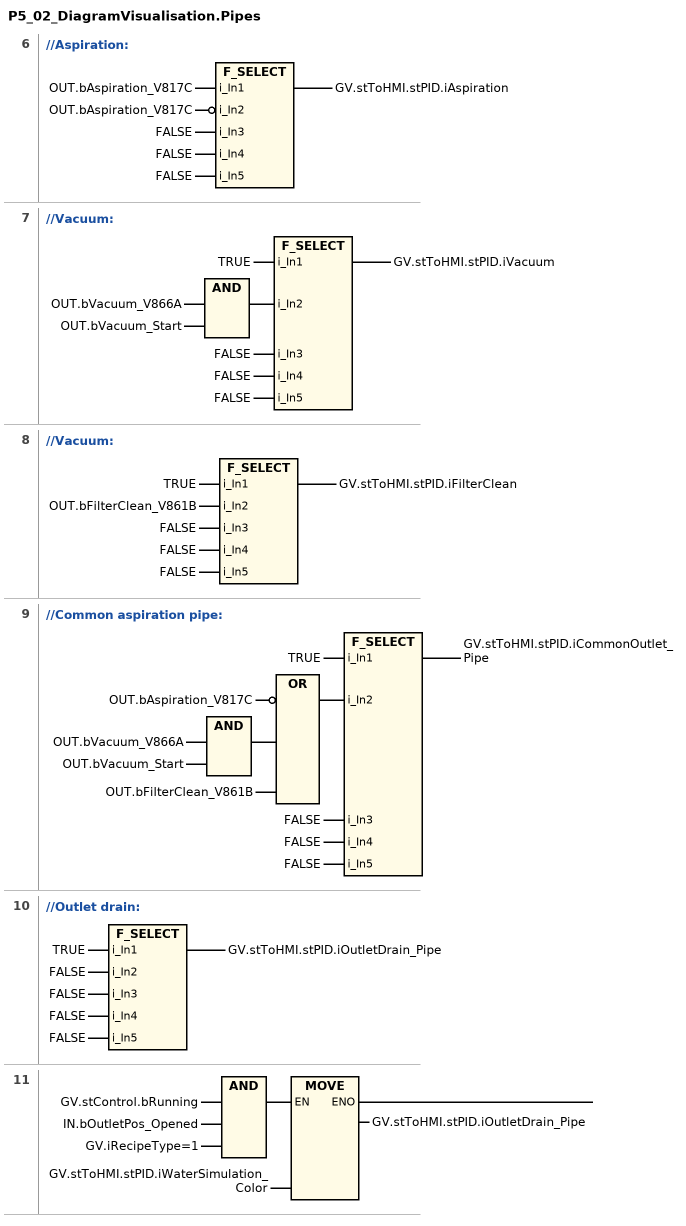
// NETWORK 6
// label: //Aspiration
GV.stToHMI.stPID.iAspiration := F_SELECT(i_In1 := OUT.bAspiration_V817C, i_In2 := NOT OUT.bAspiration_V817C, i_In3 := FALSE, i_In4 := FALSE, i_In5 := FALSE);

// NETWORK 7
// label: //Vacuum
GV.stToHMI.stPID.iVacuum := F_SELECT(i_In1 := TRUE, i_In2 := OUT.bVacuum_V866A AND OUT.bVacuum_Start, i_In3 := FALSE, i_In4 := FALSE, i_In5 := FALSE);

// NETWORK 8
// label: //Vacuum
GV.stToHMI.stPID.iFilterClean := F_SELECT(i_In1 := TRUE, i_In2 := OUT.bFilterClean_V861B, i_In3 := FALSE, i_In4 := FALSE, i_In5 := FALSE);

// NETWORK 9
// label: //Common aspiration pipe
GV.stToHMI.stPID.iCommonOutlet_Pipe := F_SELECT(i_In1 := TRUE, i_In2 := NOT OUT.bAspiration_V817C OR OUT.bVacuum_V866A AND OUT.bVacuum_Start OR OUT.bFilterClean_V861B, i_In3 := FALSE, i_In4 := FALSE, i_In5 := FALSE);

// NETWORK 10
// label: //Outlet drain
GV.stToHMI.stPID.iOutletDrain_Pipe := F_SELECT(i_In1 := TRUE, i_In2 := FALSE, i_In3 := FALSE, i_In4 := FALSE, i_In5 := FALSE);

// NETWORK 11
IF GV.stControl.bRunning AND IN.bOutletPos_Opened AND (GV.iRecipeType=1) THEN
    GV.stToHMI.stPID.iOutletDrain_Pipe := GV.stToHMI.stPID.iWaterSimulation_Color;
END_IF

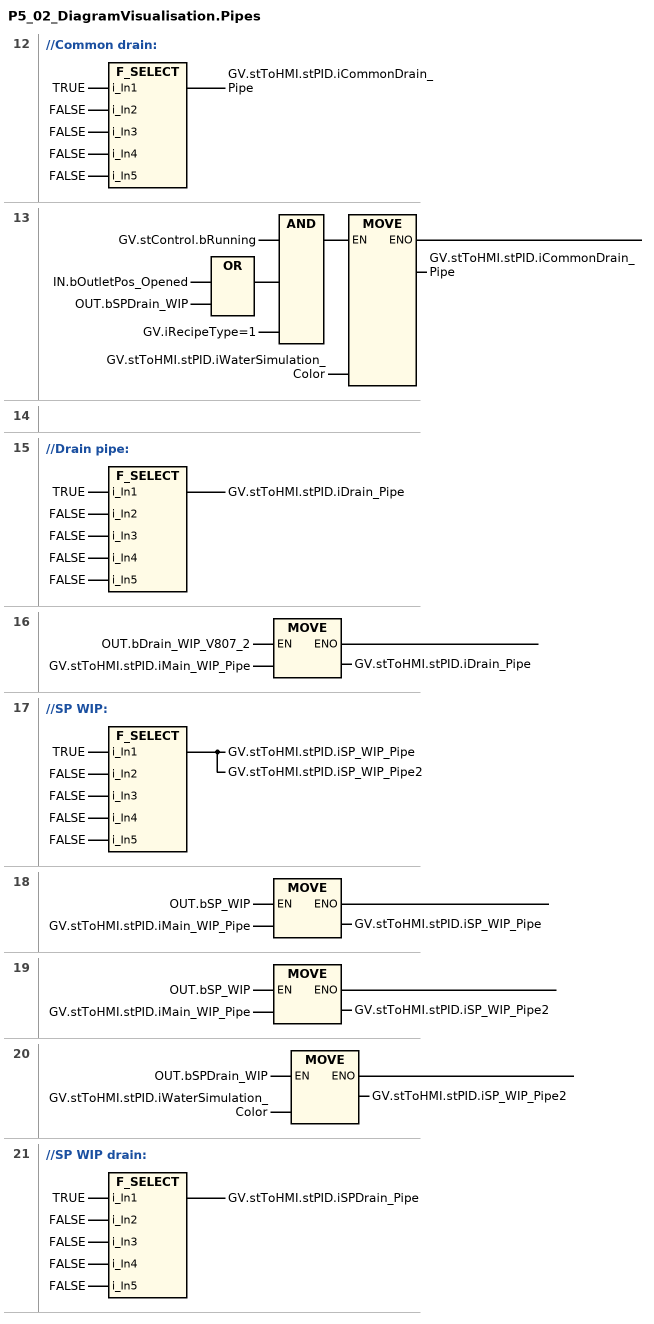
// NETWORK 12
// label: //Common drain
GV.stToHMI.stPID.iCommonDrain_Pipe := F_SELECT(i_In1 := TRUE, i_In2 := FALSE, i_In3 := FALSE, i_In4 := FALSE, i_In5 := FALSE);

// NETWORK 13
IF GV.stControl.bRunning AND (IN.bOutletPos_Opened OR OUT.bSPDrain_WIP) AND (GV.iRecipeType=1) THEN
    GV.stToHMI.stPID.iCommonDrain_Pipe := GV.stToHMI.stPID.iWaterSimulation_Color;
END_IF

// NETWORK 14

// NETWORK 15
// label: //Drain pipe
GV.stToHMI.stPID.iDrain_Pipe := F_SELECT(i_In1 := TRUE, i_In2 := FALSE, i_In3 := FALSE, i_In4 := FALSE, i_In5 := FALSE);

// NETWORK 16
IF OUT.bDrain_WIP_V807_2 THEN GV.stToHMI.stPID.iDrain_Pipe := GV.stToHMI.stPID.iMain_WIP_Pipe; END_IF

// NETWORK 17
// label: //SP WIP
_w4 := F_SELECT(i_In1 := TRUE, i_In2 := FALSE, i_In3 := FALSE, i_In4 := FALSE, i_In5 := FALSE);
GV.stToHMI.stPID.iSP_WIP_Pipe := _w4;
GV.stToHMI.stPID.iSP_WIP_Pipe2 := _w4;

// NETWORK 18
IF OUT.bSP_WIP THEN GV.stToHMI.stPID.iSP_WIP_Pipe := GV.stToHMI.stPID.iMain_WIP_Pipe; END_IF

// NETWORK 19
IF OUT.bSP_WIP THEN GV.stToHMI.stPID.iSP_WIP_Pipe2 := GV.stToHMI.stPID.iMain_WIP_Pipe; END_IF

// NETWORK 20
IF OUT.bSPDrain_WIP THEN GV.stToHMI.stPID.iSP_WIP_Pipe2 := GV.stToHMI.stPID.iWaterSimulation_Color; END_IF

// NETWORK 21
// label: //SP WIP drain
GV.stToHMI.stPID.iSPDrain_Pipe := F_SELECT(i_In1 := TRUE, i_In2 := FALSE, i_In3 := FALSE, i_In4 := FALSE, i_In5 := FALSE);

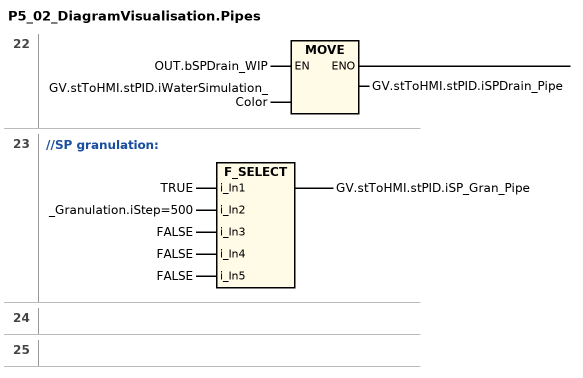
// NETWORK 22
IF OUT.bSPDrain_WIP THEN GV.stToHMI.stPID.iSPDrain_Pipe := GV.stToHMI.stPID.iWaterSimulation_Color; END_IF

// NETWORK 23
// label: //SP granulation
GV.stToHMI.stPID.iSP_Gran_Pipe := F_SELECT(i_In1 := TRUE, i_In2 := _Granulation.iStep=500, i_In3 := FALSE, i_In4 := FALSE, i_In5 := FALSE);

// NETWORK 24

// NETWORK 25
END_ACTION

ACTION Sensors:
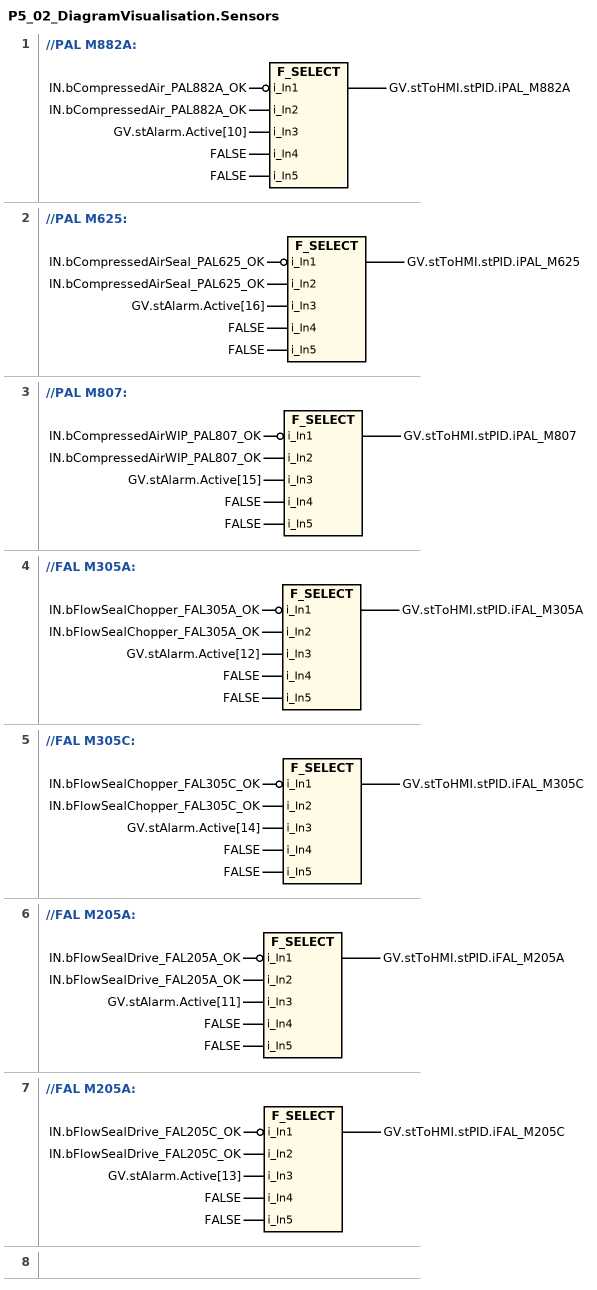
// NETWORK 1
// label: //PAL M882A
GV.stToHMI.stPID.iPAL_M882A := F_SELECT(i_In1 := NOT IN.bCompressedAir_PAL882A_OK, i_In2 := IN.bCompressedAir_PAL882A_OK, i_In3 := GV.stAlarm.Active[10], i_In4 := FALSE, i_In5 := FALSE);

// NETWORK 2
// label: //PAL M625
GV.stToHMI.stPID.iPAL_M625 := F_SELECT(i_In1 := NOT IN.bCompressedAirSeal_PAL625_OK, i_In2 := IN.bCompressedAirSeal_PAL625_OK, i_In3 := GV.stAlarm.Active[16], i_In4 := FALSE, i_In5 := FALSE);

// NETWORK 3
// label: //PAL M807
GV.stToHMI.stPID.iPAL_M807 := F_SELECT(i_In1 := NOT IN.bCompressedAirWIP_PAL807_OK, i_In2 := IN.bCompressedAirWIP_PAL807_OK, i_In3 := GV.stAlarm.Active[15], i_In4 := FALSE, i_In5 := FALSE);

// NETWORK 4
// label: //FAL M305A
GV.stToHMI.stPID.iFAL_M305A := F_SELECT(i_In1 := NOT IN.bFlowSealChopper_FAL305A_OK, i_In2 := IN.bFlowSealChopper_FAL305A_OK, i_In3 := GV.stAlarm.Active[12], i_In4 := FALSE, i_In5 := FALSE);

// NETWORK 5
// label: //FAL M305C
GV.stToHMI.stPID.iFAL_M305C := F_SELECT(i_In1 := NOT IN.bFlowSealChopper_FAL305C_OK, i_In2 := IN.bFlowSealChopper_FAL305C_OK, i_In3 := GV.stAlarm.Active[14], i_In4 := FALSE, i_In5 := FALSE);

// NETWORK 6
// label: //FAL M205A
GV.stToHMI.stPID.iFAL_M205A := F_SELECT(i_In1 := NOT IN.bFlowSealDrive_FAL205A_OK, i_In2 := IN.bFlowSealDrive_FAL205A_OK, i_In3 := GV.stAlarm.Active[11], i_In4 := FALSE, i_In5 := FALSE);

// NETWORK 7
// label: //FAL M205A
GV.stToHMI.stPID.iFAL_M205C := F_SELECT(i_In1 := NOT IN.bFlowSealDrive_FAL205C_OK, i_In2 := IN.bFlowSealDrive_FAL205C_OK, i_In3 := GV.stAlarm.Active[13], i_In4 := FALSE, i_In5 := FALSE);

// NETWORK 8
END_ACTION

ACTION Units:
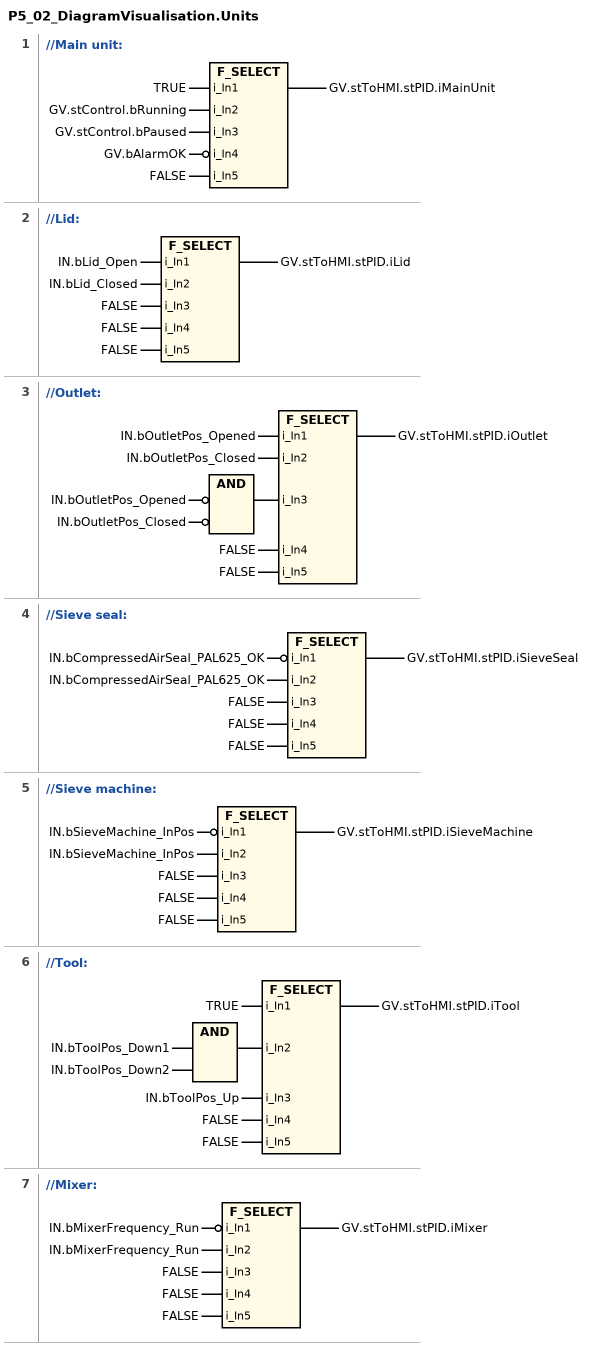
// NETWORK 1
// label: //Main unit
GV.stToHMI.stPID.iMainUnit := F_SELECT(i_In1 := TRUE, i_In2 := GV.stControl.bRunning, i_In3 := GV.stControl.bPaused, i_In4 := NOT GV.bAlarmOK, i_In5 := FALSE);

// NETWORK 2
// label: //Lid
GV.stToHMI.stPID.iLid := F_SELECT(i_In1 := IN.bLid_Open, i_In2 := IN.bLid_Closed, i_In3 := FALSE, i_In4 := FALSE, i_In5 := FALSE);

// NETWORK 3
// label: //Outlet
GV.stToHMI.stPID.iOutlet := F_SELECT(i_In1 := IN.bOutletPos_Opened, i_In2 := IN.bOutletPos_Closed, i_In3 := NOT IN.bOutletPos_Opened AND NOT IN.bOutletPos_Closed, i_In4 := FALSE, i_In5 := FALSE);

// NETWORK 4
// label: //Sieve seal
GV.stToHMI.stPID.iSieveSeal := F_SELECT(i_In1 := NOT IN.bCompressedAirSeal_PAL625_OK, i_In2 := IN.bCompressedAirSeal_PAL625_OK, i_In3 := FALSE, i_In4 := FALSE, i_In5 := FALSE);

// NETWORK 5
// label: //Sieve machine
GV.stToHMI.stPID.iSieveMachine := F_SELECT(i_In1 := NOT IN.bSieveMachine_InPos, i_In2 := IN.bSieveMachine_InPos, i_In3 := FALSE, i_In4 := FALSE, i_In5 := FALSE);

// NETWORK 6
// label: //Tool
GV.stToHMI.stPID.iTool := F_SELECT(i_In1 := TRUE, i_In2 := IN.bToolPos_Down1 AND IN.bToolPos_Down2, i_In3 := IN.bToolPos_Up, i_In4 := FALSE, i_In5 := FALSE);

// NETWORK 7
// label: //Mixer
GV.stToHMI.stPID.iMixer := F_SELECT(i_In1 := NOT IN.bMixerFrequency_Run, i_In2 := IN.bMixerFrequency_Run, i_In3 := FALSE, i_In4 := FALSE, i_In5 := FALSE);

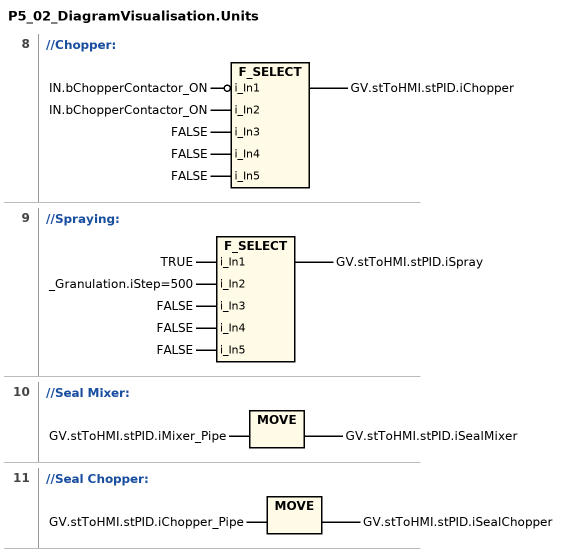
// NETWORK 8
// label: //Chopper
GV.stToHMI.stPID.iChopper := F_SELECT(i_In1 := NOT IN.bChopperContactor_ON, i_In2 := IN.bChopperContactor_ON, i_In3 := FALSE, i_In4 := FALSE, i_In5 := FALSE);

// NETWORK 9
// label: //Spraying
GV.stToHMI.stPID.iSpray := F_SELECT(i_In1 := TRUE, i_In2 := _Granulation.iStep=500, i_In3 := FALSE, i_In4 := FALSE, i_In5 := FALSE);

// NETWORK 10
// label: //Seal Mixer
GV.stToHMI.stPID.iSealMixer := GV.stToHMI.stPID.iMixer_Pipe;

// NETWORK 11
// label: //Seal Chopper
GV.stToHMI.stPID.iSealChopper := GV.stToHMI.stPID.iChopper_Pipe;
END_ACTION

END_PROGRAM

// ---- Functions/F_Select.TcPOU
FUNCTION F_Select : INT
VAR_INPUT
	i_In1			:BOOL;
	i_In2			:BOOL;
	i_In3			:BOOL;
	i_In4			:BOOL;
	i_In5			:BOOL;
END_VAR
VAR
END_VAR

IF i_In1 THEN
	F_Select:=0;
END_IF
IF i_In2 THEN
	F_Select:=1;
END_IF
IF i_In3 THEN
	F_Select:=2;
END_IF
IF i_In4 THEN
	F_Select:=3;
END_IF
IF i_In5 THEN
	F_Select:=4;
END_IF

END_FUNCTION

// ---- POUs/5. HMI/P5_03_OtherControl.TcPOU
PROGRAM P5_03_OtherControl
VAR
	iSeqControl				:INT;
	tSubStepET				:TIME;
	tSubStepPT				:TIME;
	iSubStepMC				:INT;
	iSubStepPC				:INT;
END_VAR
VAR // added by the converter: edge detectors and wires of the graphical bodies
    _w1, _w2 : TIME;
    _w3, _w4 : BOOL;
END_VAR

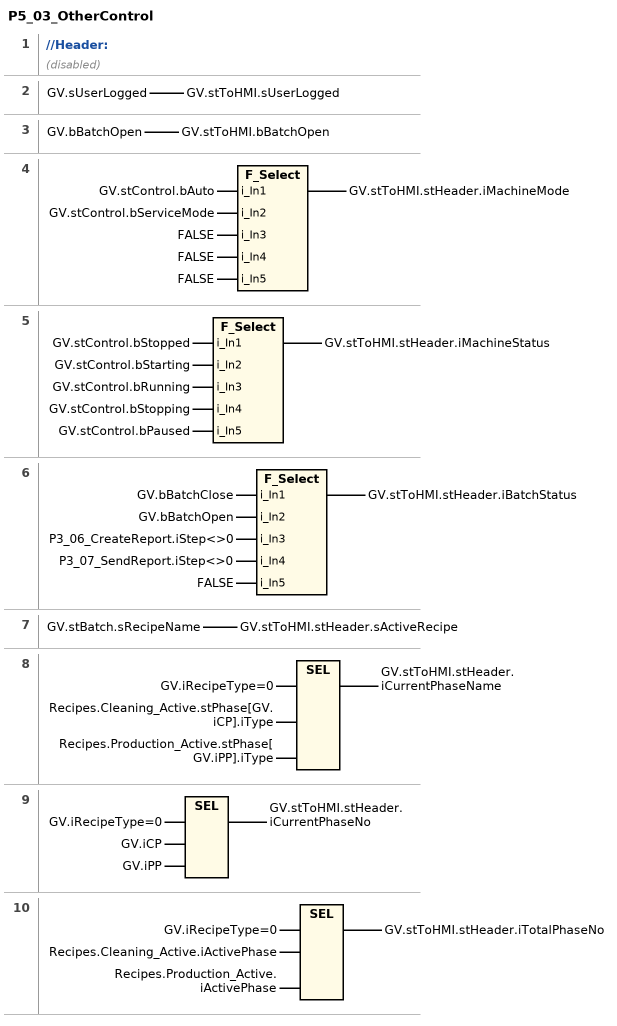
// NETWORK 1 (disabled)
// label: //Header

// NETWORK 2
GV.stToHMI.sUserLogged := GV.sUserLogged;

// NETWORK 3
GV.stToHMI.bBatchOpen := GV.bBatchOpen;

// NETWORK 4
GV.stToHMI.stHeader.iMachineMode := F_Select(i_In1 := GV.stControl.bAuto, i_In2 := GV.stControl.bServiceMode, i_In3 := FALSE, i_In4 := FALSE, i_In5 := FALSE);

// NETWORK 5
GV.stToHMI.stHeader.iMachineStatus := F_Select(i_In1 := GV.stControl.bStopped, i_In2 := GV.stControl.bStarting, i_In3 := GV.stControl.bRunning, i_In4 := GV.stControl.bStopping, i_In5 := GV.stControl.bPaused);

// NETWORK 6
GV.stToHMI.stHeader.iBatchStatus := F_Select(i_In1 := GV.bBatchClose, i_In2 := GV.bBatchOpen, i_In3 := P3_06_CreateReport.iStep<>0, i_In4 := P3_07_SendReport.iStep<>0, i_In5 := FALSE);

// NETWORK 7
GV.stToHMI.stHeader.sActiveRecipe := GV.stBatch.sRecipeName;

// NETWORK 8
GV.stToHMI.stHeader.iCurrentPhaseName := SEL(GV.iRecipeType=0, Recipes.Cleaning_Active.stPhase[GV.iCP].iType, Recipes.Production_Active.stPhase[GV.iPP].iType);

// NETWORK 9
GV.stToHMI.stHeader.iCurrentPhaseNo := SEL(GV.iRecipeType=0, GV.iCP, GV.iPP);

// NETWORK 10
GV.stToHMI.stHeader.iTotalPhaseNo := SEL(GV.iRecipeType=0, Recipes.Cleaning_Active.iActivePhase, Recipes.Production_Active.iActivePhase);

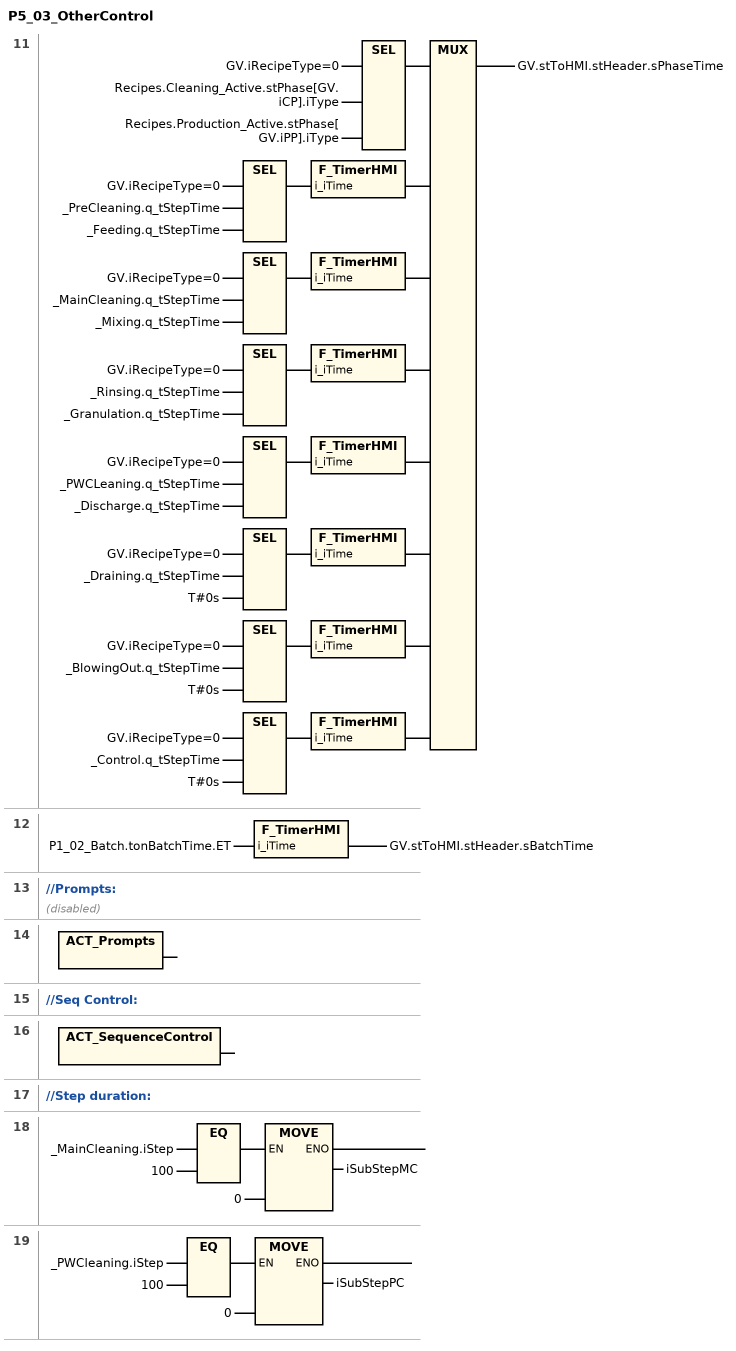
// NETWORK 11
GV.stToHMI.stHeader.sPhaseTime := MUX(SEL(GV.iRecipeType=0, Recipes.Cleaning_Active.stPhase[GV.iCP].iType, Recipes.Production_Active.stPhase[GV.iPP].iType), F_TimerHMI(i_iTime := SEL(GV.iRecipeType=0, _PreCleaning.q_tStepTime, _Feeding.q_tStepTime)), F_TimerHMI(i_iTime := SEL(GV.iRecipeType=0, _MainCleaning.q_tStepTime, _Mixing.q_tStepTime)), F_TimerHMI(i_iTime := SEL(GV.iRecipeType=0, _Rinsing.q_tStepTime, _Granulation.q_tStepTime)), F_TimerHMI(i_iTime := SEL(GV.iRecipeType=0, _PWCLeaning.q_tStepTime, _Discharge.q_tStepTime)), F_TimerHMI(i_iTime := SEL(GV.iRecipeType=0, _Draining.q_tStepTime, T#0s)), F_TimerHMI(i_iTime := SEL(GV.iRecipeType=0, _BlowingOut.q_tStepTime, T#0s)), F_TimerHMI(i_iTime := SEL(GV.iRecipeType=0, _Control.q_tStepTime, T#0s)));

// NETWORK 12
GV.stToHMI.stHeader.sBatchTime := F_TimerHMI(i_iTime := P1_02_Batch.tonBatchTime.ET);

// NETWORK 13 (disabled)
// label: //Prompts

// NETWORK 14
ACT_Prompts();

// NETWORK 15
// label: //Seq Control

// NETWORK 16
ACT_SequenceControl();

// NETWORK 17
// label: //Step duration

// NETWORK 18
IF _MainCleaning.iStep = 100 THEN iSubStepMC := 0; END_IF

// NETWORK 19
IF _PWCleaning.iStep = 100 THEN iSubStepPC := 0; END_IF

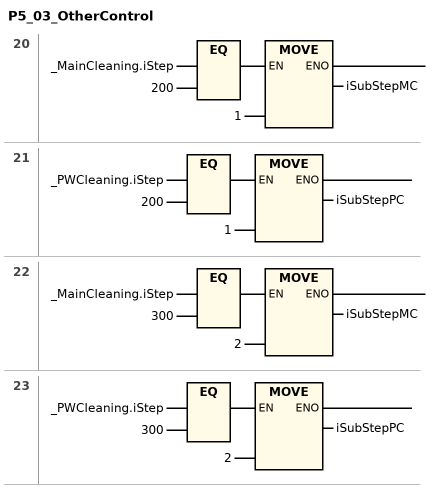
// NETWORK 20
IF _MainCleaning.iStep = 200 THEN iSubStepMC := 1; END_IF

// NETWORK 21
IF _PWCleaning.iStep = 200 THEN iSubStepPC := 1; END_IF

// NETWORK 22
IF _MainCleaning.iStep = 300 THEN iSubStepMC := 2; END_IF

// NETWORK 23
IF _PWCleaning.iStep = 300 THEN iSubStepPC := 2; END_IF

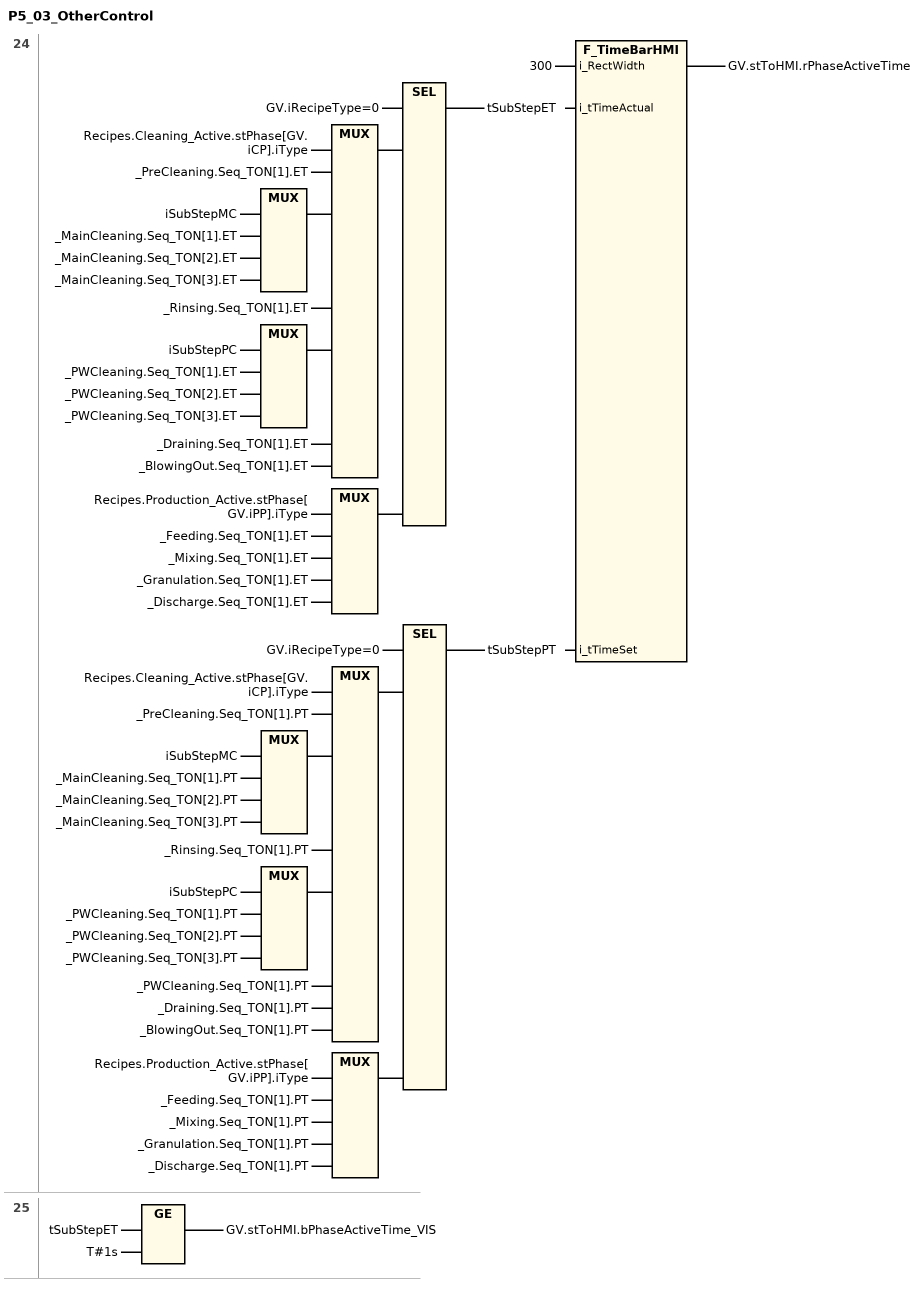
// NETWORK 24
_w1 := SEL(GV.iRecipeType=0, MUX(Recipes.Cleaning_Active.stPhase[GV.iCP].iType, _PreCleaning.Seq_TON[1].ET, MUX(iSubStepMC, _MainCleaning.Seq_TON[1].ET, _MainCleaning.Seq_TON[2].ET, _MainCleaning.Seq_TON[3].ET), _Rinsing.Seq_TON[1].ET, MUX(iSubStepPC, _PWCleaning.Seq_TON[1].ET, _PWCleaning.Seq_TON[2].ET, _PWCleaning.Seq_TON[3].ET), _Draining.Seq_TON[1].ET, _BlowingOut.Seq_TON[1].ET), MUX(Recipes.Production_Active.stPhase[GV.iPP].iType, _Feeding.Seq_TON[1].ET, _Mixing.Seq_TON[1].ET, _Granulation.Seq_TON[1].ET, _Discharge.Seq_TON[1].ET));
tSubStepET := _w1;
_w2 := SEL(GV.iRecipeType=0, MUX(Recipes.Cleaning_Active.stPhase[GV.iCP].iType, _PreCleaning.Seq_TON[1].PT, MUX(iSubStepMC, _MainCleaning.Seq_TON[1].PT, _MainCleaning.Seq_TON[2].PT, _MainCleaning.Seq_TON[3].PT), _Rinsing.Seq_TON[1].PT, MUX(iSubStepPC, _PWCleaning.Seq_TON[1].PT, _PWCleaning.Seq_TON[2].PT, _PWCleaning.Seq_TON[3].PT), _PWCleaning.Seq_TON[1].PT, _Draining.Seq_TON[1].PT, _BlowingOut.Seq_TON[1].PT), MUX(Recipes.Production_Active.stPhase[GV.iPP].iType, _Feeding.Seq_TON[1].PT, _Mixing.Seq_TON[1].PT, _Granulation.Seq_TON[1].PT, _Discharge.Seq_TON[1].PT));
tSubStepPT := _w2;
GV.stToHMI.rPhaseActiveTime := F_TimeBarHMI(i_RectWidth := 300, i_tTimeActual := _w1, i_tTimeSet := _w2);

// NETWORK 25
GV.stToHMI.bPhaseActiveTime_VIS := tSubStepET >= T#1s;

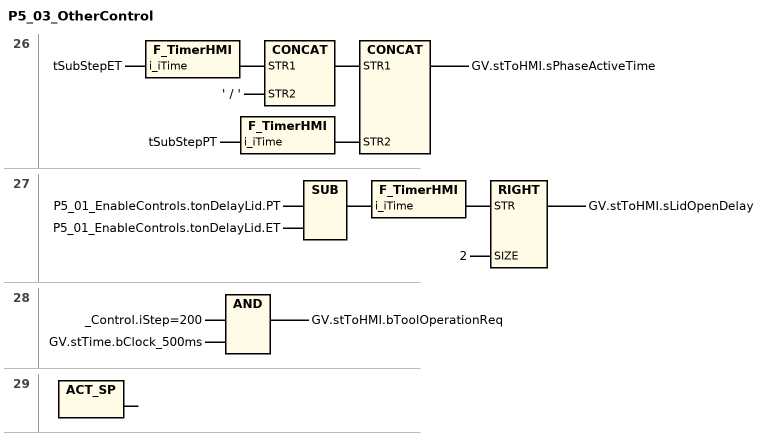
// NETWORK 26
GV.stToHMI.sPhaseActiveTime := CONCAT(STR1 := CONCAT(STR1 := F_TimerHMI(i_iTime := tSubStepET), STR2 := ' / '), STR2 := F_TimerHMI(i_iTime := tSubStepPT));

// NETWORK 27
GV.stToHMI.sLidOpenDelay := RIGHT(STR := F_TimerHMI(i_iTime := P5_01_EnableControls.tonDelayLid.PT - P5_01_EnableControls.tonDelayLid.ET), SIZE := 2);

// NETWORK 28
GV.stToHMI.bToolOperationReq := (_Control.iStep=200) AND GV.stTime.bClock_500ms;

// NETWORK 29
ACT_SP();

ACTION ACT_Prompts:
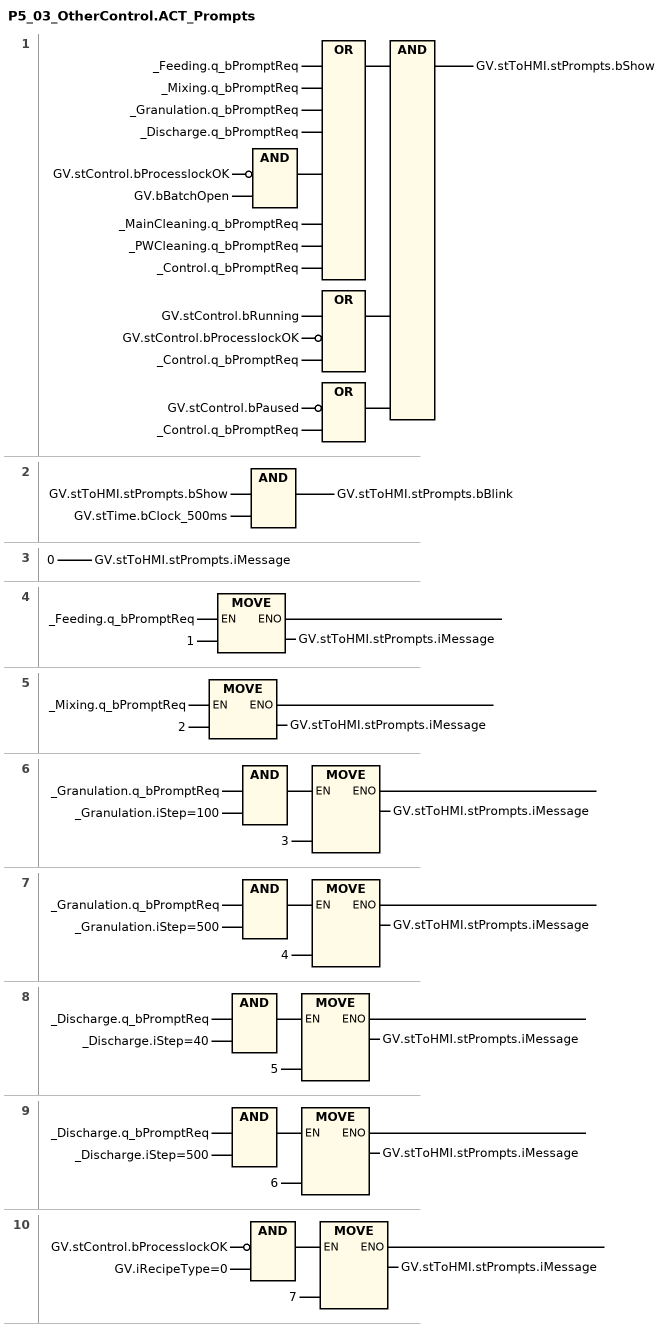
// NETWORK 1
GV.stToHMI.stPrompts.bShow := (_Feeding.q_bPromptReq OR _Mixing.q_bPromptReq OR _Granulation.q_bPromptReq OR _Discharge.q_bPromptReq OR NOT GV.stControl.bProcesslockOK AND GV.bBatchOpen OR _MainCleaning.q_bPromptReq OR _PWCleaning.q_bPromptReq OR _Control.q_bPromptReq) AND (GV.stControl.bRunning OR NOT GV.stControl.bProcesslockOK OR _Control.q_bPromptReq) AND (NOT GV.stControl.bPaused OR _Control.q_bPromptReq);

// NETWORK 2
GV.stToHMI.stPrompts.bBlink := GV.stToHMI.stPrompts.bShow AND GV.stTime.bClock_500ms;

// NETWORK 3
GV.stToHMI.stPrompts.iMessage := 0;

// NETWORK 4
IF _Feeding.q_bPromptReq THEN GV.stToHMI.stPrompts.iMessage := 1; END_IF

// NETWORK 5
IF _Mixing.q_bPromptReq THEN GV.stToHMI.stPrompts.iMessage := 2; END_IF

// NETWORK 6
IF _Granulation.q_bPromptReq AND (_Granulation.iStep=100) THEN GV.stToHMI.stPrompts.iMessage := 3; END_IF

// NETWORK 7
IF _Granulation.q_bPromptReq AND (_Granulation.iStep=500) THEN GV.stToHMI.stPrompts.iMessage := 4; END_IF

// NETWORK 8
IF _Discharge.q_bPromptReq AND (_Discharge.iStep=40) THEN GV.stToHMI.stPrompts.iMessage := 5; END_IF

// NETWORK 9
IF _Discharge.q_bPromptReq AND (_Discharge.iStep=500) THEN GV.stToHMI.stPrompts.iMessage := 6; END_IF

// NETWORK 10
IF NOT GV.stControl.bProcesslockOK AND (GV.iRecipeType=0) THEN GV.stToHMI.stPrompts.iMessage := 7; END_IF

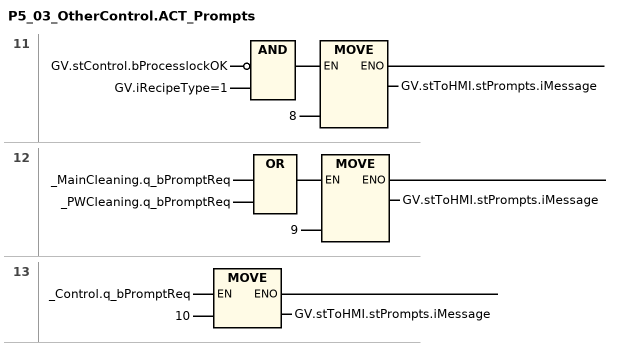
// NETWORK 11
IF NOT GV.stControl.bProcesslockOK AND (GV.iRecipeType=1) THEN GV.stToHMI.stPrompts.iMessage := 8; END_IF

// NETWORK 12
IF _MainCleaning.q_bPromptReq OR _PWCleaning.q_bPromptReq THEN GV.stToHMI.stPrompts.iMessage := 9; END_IF

// NETWORK 13
IF _Control.q_bPromptReq THEN GV.stToHMI.stPrompts.iMessage := 10; END_IF
END_ACTION

ACTION ACT_SequenceControl:
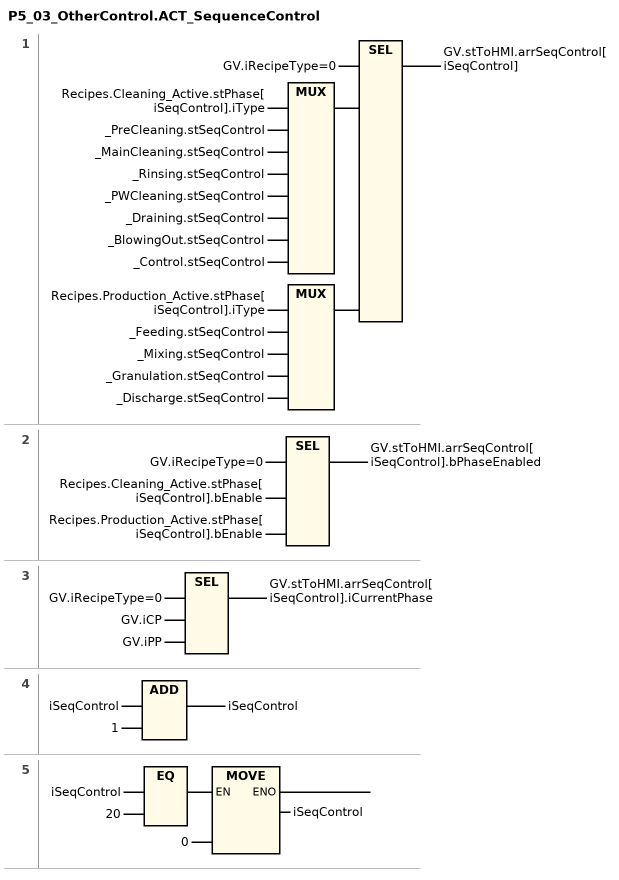
// NETWORK 1
GV.stToHMI.arrSeqControl[iSeqControl] := SEL(GV.iRecipeType=0, MUX(Recipes.Cleaning_Active.stPhase[iSeqControl].iType, _PreCleaning.stSeqControl, _MainCleaning.stSeqControl, _Rinsing.stSeqControl, _PWCleaning.stSeqControl, _Draining.stSeqControl, _BlowingOut.stSeqControl, _Control.stSeqControl), MUX(Recipes.Production_Active.stPhase[iSeqControl].iType, _Feeding.stSeqControl, _Mixing.stSeqControl, _Granulation.stSeqControl, _Discharge.stSeqControl));

// NETWORK 2
GV.stToHMI.arrSeqControl[iSeqControl].bPhaseEnabled := SEL(GV.iRecipeType=0, Recipes.Cleaning_Active.stPhase[iSeqControl].bEnable, Recipes.Production_Active.stPhase[iSeqControl].bEnable);

// NETWORK 3
GV.stToHMI.arrSeqControl[iSeqControl].iCurrentPhase := SEL(GV.iRecipeType=0, GV.iCP, GV.iPP);

// NETWORK 4
iSeqControl := iSeqControl + 1;

// NETWORK 5
IF iSeqControl = 20 THEN iSeqControl := 0; END_IF
END_ACTION

ACTION ACT_SP:
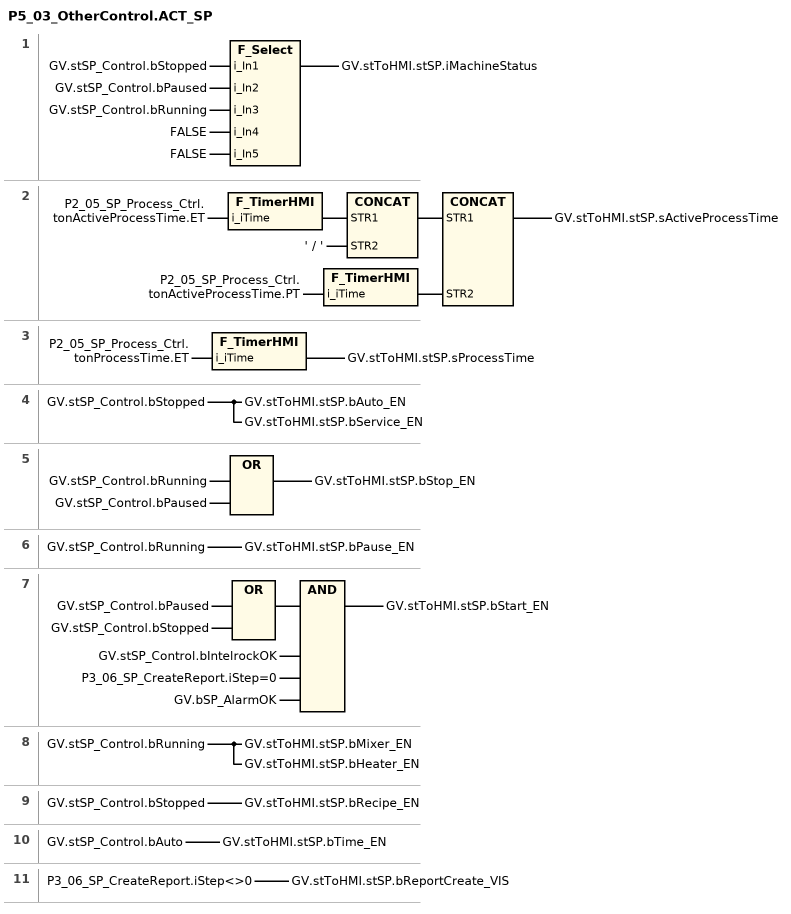
// NETWORK 1
GV.stToHMI.stSP.iMachineStatus := F_Select(i_In1 := GV.stSP_Control.bStopped, i_In2 := GV.stSP_Control.bPaused, i_In3 := GV.stSP_Control.bRunning, i_In4 := FALSE, i_In5 := FALSE);

// NETWORK 2
GV.stToHMI.stSP.sActiveProcessTime := CONCAT(STR1 := CONCAT(STR1 := F_TimerHMI(i_iTime := P2_05_SP_Process_Ctrl.tonActiveProcessTime.ET), STR2 := ' / '), STR2 := F_TimerHMI(i_iTime := P2_05_SP_Process_Ctrl.tonActiveProcessTime.PT));

// NETWORK 3
GV.stToHMI.stSP.sProcessTime := F_TimerHMI(i_iTime := P2_05_SP_Process_Ctrl.tonProcessTime.ET);

// NETWORK 4
_w3 := GV.stSP_Control.bStopped;
GV.stToHMI.stSP.bAuto_EN := _w3;
GV.stToHMI.stSP.bService_EN := _w3;

// NETWORK 5
GV.stToHMI.stSP.bStop_EN := GV.stSP_Control.bRunning OR GV.stSP_Control.bPaused;

// NETWORK 6
GV.stToHMI.stSP.bPause_EN := GV.stSP_Control.bRunning;

// NETWORK 7
GV.stToHMI.stSP.bStart_EN := (GV.stSP_Control.bPaused OR GV.stSP_Control.bStopped) AND GV.stSP_Control.bIntelrockOK AND (P3_06_SP_CreateReport.iStep=0) AND GV.bSP_AlarmOK;

// NETWORK 8
_w4 := GV.stSP_Control.bRunning;
GV.stToHMI.stSP.bMixer_EN := _w4;
GV.stToHMI.stSP.bHeater_EN := _w4;

// NETWORK 9
GV.stToHMI.stSP.bRecipe_EN := GV.stSP_Control.bStopped;

// NETWORK 10
GV.stToHMI.stSP.bTime_EN := GV.stSP_Control.bAuto;

// NETWORK 11
GV.stToHMI.stSP.bReportCreate_VIS := P3_06_SP_CreateReport.iStep<>0;
END_ACTION

END_PROGRAM

// ---- POUs/5. HMI/P5_04_Trends.TcPOU
PROGRAM P5_04_Trends
VAR
END_VAR

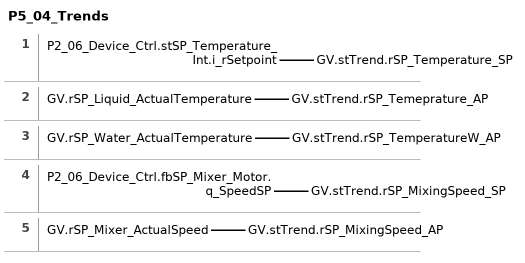
// NETWORK 1
GV.stTrend.rSP_Temperature_SP := P2_06_Device_Ctrl.stSP_Temperature_Int.i_rSetpoint;

// NETWORK 2
GV.stTrend.rSP_Temeprature_AP := GV.rSP_Liquid_ActualTemperature;

// NETWORK 3
GV.stTrend.rSP_TemperatureW_AP := GV.rSP_Water_ActualTemperature;

// NETWORK 4
GV.stTrend.rSP_MixingSpeed_SP := P2_06_Device_Ctrl.fbSP_Mixer_Motor.q_SpeedSP;

// NETWORK 5
GV.stTrend.rSP_MixingSpeed_AP := GV.rSP_Mixer_ActualSpeed;

END_PROGRAM

// ---- POUs/SIMULATION.TcPOU
PROGRAM SIMULATION
VAR
	TON_0: TON;
	TON_1: TON;
	TON_2: TON;
	TON_3: TON;
	TON_4: TON;
	bPAL_M882A			:BOOL:=TRUE;
	TON_5: TON;
	TON_6: TON;
	TON_7: TON;
	TON_8: TON;
	
	rMixerAngle			:REAL;
	iRevolutions		:INT;
	tonMixerRPM			:TON;
	fbScaleMixerRev		:FB_Scale;
END_VAR


VAR PERSISTENT
	TIME_5: TIME;
	TIME_6: TIME;
END_VAR
VAR // added by the converter: edge detectors and wires of the graphical bodies
    _w1, _w2, _w3 : BOOL;
END_VAR

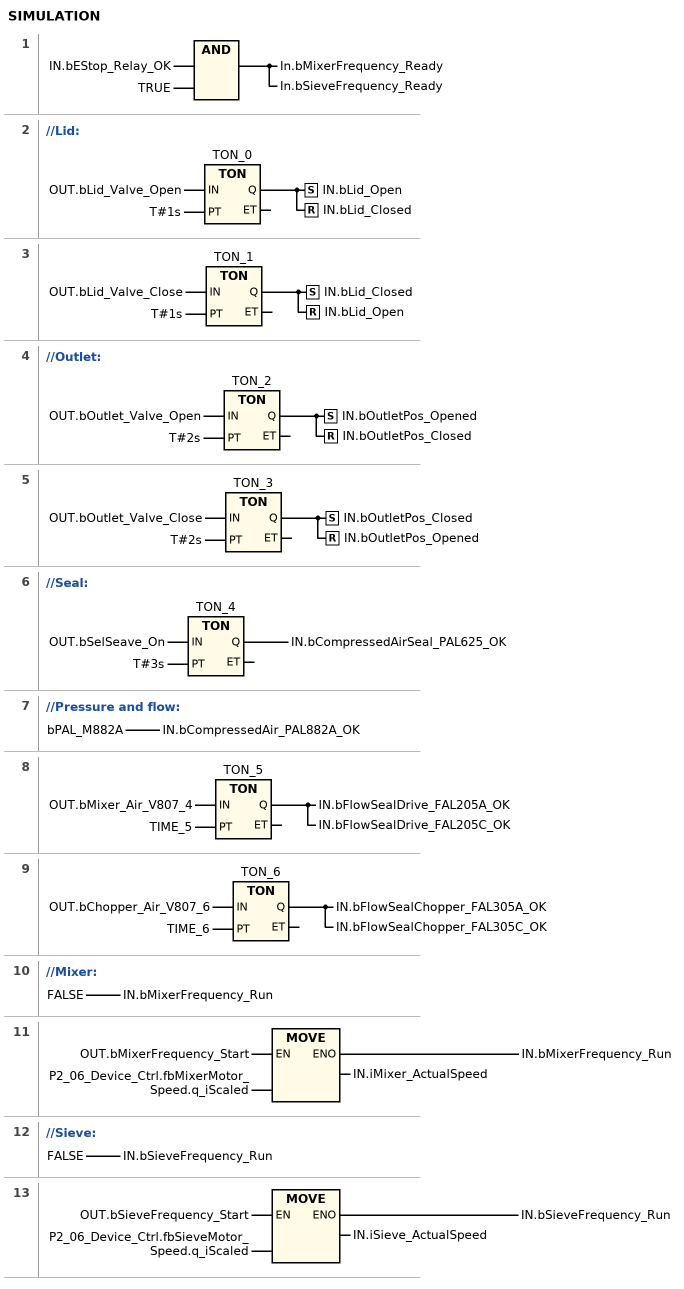
// NETWORK 1
_w1 := IN.bEStop_Relay_OK AND TRUE;
In.bMixerFrequency_Ready := _w1;
In.bSieveFrequency_Ready := _w1;

// NETWORK 2
// label: //Lid
TON_0(IN := OUT.bLid_Valve_Open, PT := T#1s); // TON
IN.bLid_Open S= TON_0.Q;
IN.bLid_Closed R= TON_0.Q;

// NETWORK 3
TON_1(IN := OUT.bLid_Valve_Close, PT := T#1s); // TON
IN.bLid_Closed S= TON_1.Q;
IN.bLid_Open R= TON_1.Q;

// NETWORK 4
// label: //Outlet
TON_2(IN := OUT.bOutlet_Valve_Open, PT := T#2s); // TON
IN.bOutletPos_Opened S= TON_2.Q;
IN.bOutletPos_Closed R= TON_2.Q;

// NETWORK 5
TON_3(IN := OUT.bOutlet_Valve_Close, PT := T#2s); // TON
IN.bOutletPos_Closed S= TON_3.Q;
IN.bOutletPos_Opened R= TON_3.Q;

// NETWORK 6
// label: //Seal
TON_4(IN := OUT.bSelSeave_On, PT := T#3s); // TON
IN.bCompressedAirSeal_PAL625_OK := TON_4.Q;

// NETWORK 7
// label: //Pressure and flow
IN.bCompressedAir_PAL882A_OK := bPAL_M882A;

// NETWORK 8
TON_5(IN := OUT.bMixer_Air_V807_4, PT := TIME_5); // TON
IN.bFlowSealDrive_FAL205A_OK := TON_5.Q;
IN.bFlowSealDrive_FAL205C_OK := TON_5.Q;

// NETWORK 9
TON_6(IN := OUT.bChopper_Air_V807_6, PT := TIME_6); // TON
IN.bFlowSealChopper_FAL305A_OK := TON_6.Q;
IN.bFlowSealChopper_FAL305C_OK := TON_6.Q;

// NETWORK 10
// label: //Mixer
IN.bMixerFrequency_Run := FALSE;

// NETWORK 11
_w2 := OUT.bMixerFrequency_Start;
IF _w2 THEN IN.iMixer_ActualSpeed := P2_06_Device_Ctrl.fbMixerMotor_Speed.q_iScaled; END_IF
IN.bMixerFrequency_Run := _w2;

// NETWORK 12
// label: //Sieve
IN.bSieveFrequency_Run := FALSE;

// NETWORK 13
_w3 := OUT.bSieveFrequency_Start;
IF _w3 THEN IN.iSieve_ActualSpeed := P2_06_Device_Ctrl.fbSieveMotor_Speed.q_iScaled; END_IF
IN.bSieveFrequency_Run := _w3;

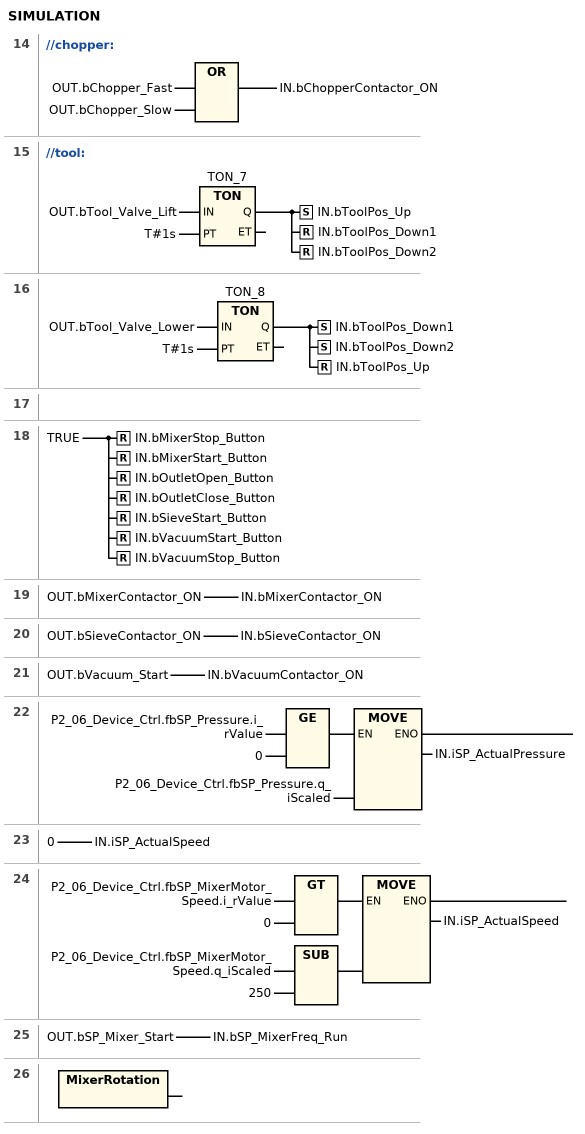
// NETWORK 14
// label: //chopper
IN.bChopperContactor_ON := OUT.bChopper_Fast OR OUT.bChopper_Slow;

// NETWORK 15
// label: //tool
TON_7(IN := OUT.bTool_Valve_Lift, PT := T#1s); // TON
IN.bToolPos_Up S= TON_7.Q;
IN.bToolPos_Down1 R= TON_7.Q;
IN.bToolPos_Down2 R= TON_7.Q;

// NETWORK 16
TON_8(IN := OUT.bTool_Valve_Lower, PT := T#1s); // TON
IN.bToolPos_Down1 S= TON_8.Q;
IN.bToolPos_Down2 S= TON_8.Q;
IN.bToolPos_Up R= TON_8.Q;

// NETWORK 17

// NETWORK 18
IN.bMixerStop_Button R= TRUE;
IN.bMixerStart_Button R= TRUE;
IN.bOutletOpen_Button R= TRUE;
IN.bOutletClose_Button R= TRUE;
IN.bSieveStart_Button R= TRUE;
IN.bVacuumStart_Button R= TRUE;
IN.bVacuumStop_Button R= TRUE;

// NETWORK 19
IN.bMixerContactor_ON := OUT.bMixerContactor_ON;

// NETWORK 20
IN.bSieveContactor_ON := OUT.bSieveContactor_ON;

// NETWORK 21
IN.bVacuumContactor_ON := OUT.bVacuum_Start;

// NETWORK 22
IF P2_06_Device_Ctrl.fbSP_Pressure.i_rValue >= 0 THEN
    IN.iSP_ActualPressure := P2_06_Device_Ctrl.fbSP_Pressure.q_iScaled;
END_IF

// NETWORK 23
IN.iSP_ActualSpeed := 0;

// NETWORK 24
IF P2_06_Device_Ctrl.fbSP_MixerMotor_Speed.i_rValue > 0 THEN
    IN.iSP_ActualSpeed := P2_06_Device_Ctrl.fbSP_MixerMotor_Speed.q_iScaled - 250;
END_IF

// NETWORK 25
IN.bSP_MixerFreq_Run := OUT.bSP_Mixer_Start;

// NETWORK 26
MixerRotation();

ACTION MixerRotation:

tonMixerRPM(IN:=P2_06_Device_Ctrl.fbMixerMotor_Speed.i_rValue<>0 AND OUT.bMixerFrequency_Start AND NOT tonMixerRPM.Q ,
			PT:=TO_TIME(P2_06_Device_Ctrl.fbMixerMotor_Speed.i_rValue/60*1000));

IF tonMixerRPM.Q THEN
	iRevolutions:=iRevolutions+1;
END_IF

IF iRevolutions > 32000 THEN
	iRevolutions:=0;
END_IF
IF TO_REAL(tonMixerRPM.PT) <> 0 THEN
	fbScaleMixerRev(i_rValue:=TO_REAL(tonMixerRPM.ET),
					i_rRawData_Low:=0,
					i_rRawData_High:=TO_REAL(tonMixerRPM.PT),
					i_rScaled_Low:=0,
					i_rScaled_High:=360,
					i_rOffset:=0,
					q_rScaled=>rMixerAngle);
END_IF	
IF rMixerAngle > 100 AND rMixerAngle < 150 THEN
	IN.bMixerTool_InPos:=TRUE;
ELSE
	IN.bMixerTool_InPos:=FALSE;
END_IF
END_ACTION

END_PROGRAM

// ---- FBs/FB_AVG200.TcPOU
//Created by Dimitar Stojanov 06.2023

//Functionality: Calculate average value of the last 200 input samples, use for analog inputs that affectc PID regulation.

FUNCTION_BLOCK FB_AVG200
VAR_INPUT
	i_rSignal			:REAL;
END_VAR
VAR_OUTPUT
	q_rSignalAvg		:REAL;
END_VAR
VAR
	arrSignals			:ARRAY[0..199] OF REAL;
	i					:INT;
	j					:INT;
	k					:INT;
	Sum					:REAL;
END_VAR

FOR k:=0 TO 198 DO
	arrSignals[k]:=arrSignals[k+1];
END_FOR
arrSignals[199]:=i_rSignal;
Sum:=0;
FOR j:=0 TO 199 DO
	Sum := Sum + arrSignals[j];
END_FOR
IF Sum <> 0 THEN
	q_rSignalAvg:=Sum/200;
ELSIF Sum = 0 THEN
	q_rSignalAvg:=0;
END_IF

END_FUNCTION_BLOCK
